(* Logix 5000 project; controller cal1615 1756-L62 rev 20.19; software revision 20.05; part 36 of 82 *)
(* tags used below, declared in another part *)
   AFI : BOOL;   // Always False Bit
   FAULT : BOOL;   // Fault AFI
   p01_recipe_active : recipe;   // Active Recipe
   p01r09_pb_global_reset : BOOL;   // System Modes PB: Global Fault Reset
   p02_dint_from_hmi : hmi_dint;
   p02_real_from_hmi : hmi_real;   // MOP HMI Iface Real from HMI
   p11r31_timer_prs : TIMER;   // Advanced Cooling Pump Pressure On Delay
   p13r30_request_cool : BOOL;   // Zone 3 Temperature Control Request Cooling
   p19_ai_prs : REAL;   // Advanced Cooling Analog Input Pressure [PSI]
   p19_ai_tc01 : REAL;   // Advanced Cooling Analog Input Control Temperature 1
   p19_ao_cv : REAL;   // Advanced Cooling Analog Output Control Valve
   p19_ao_prs_cv : REAL;   // Advanced Cooling Pressure Control AO: Control Value
   p19_di_pump : BOOL;
   p19_di_tc01_bo : BOOL;   // Advanced Cooling Digital Input Control Thermocouple 1 Failure
   p19_do_pump : BOOL;   // Advanced Cooling Digital Output Enable Pump
   p19_param_pid2_ff : REAL;
   p19_param_pid2_kd : REAL;
   p19_param_pid2_ki : REAL;
   p19_param_pid2_kp : REAL;
   p19_param_prs_dev : REAL;
   p19_param_prs_pid_ff : REAL;
   p19_param_prs_pid_kd : REAL;
   p19_param_prs_pid_ki : REAL;
   p19_param_prs_pid_kp : REAL;
   p19_param_tc01_dev : REAL;
   p19_param_zone_pressure : REAL;   // Advanced Cooling Parameter Minimum Pressusre
   p19r01 : routine;   // Advanced Cooling Main
   p19r10 : routine;   // Advanced Cooling Parameters
   p19r10_timer_warning : TIMER[4];   // Advanced Cooling Parameters Warning Delay
   p19r16_pid_temp_cv : DINT;   // Advanced Cooling Temperature Control PID Control Valve
   p19r30 : routine;   // Advanced Cooling Temperature Control
   p19r30_cv_man_sp : REAL;   // Advanced Cooling Manual Control Valve Setpoint
   p19r30_pb_auto : BOOL;   // Advanced Cooling Temmperature Control PB: Zone in Auto
   p19r30_pb_manual : BOOL;   // Advanced Cooling Temmperature Control PB: Zone in Manual
   p19r30_pb_zone_off : BOOL;   // Advanced Cooling Temmperature Control PB: Zone Off
   p19r30_pb_zone_on : BOOL;   // Advanced Cooling Temmperature Control PB: Zone On
   p19r30_permissive_run : BOOL;   // Advanced Cooling Temperature Control Permissive Run
   p19r30_pid_temp : PID;   // Advanced Cooling Temperature Control PID
   p19r30_pid_temp_pv : DINT;   // Advanced Cooling Temperature Control PID Process Variable
   p19r30_pid_temp_sp : DINT;   // Advanced Cooling Temeperature Control PID Setpoint
   p19r30_request_cool : BOOL;   // Advanced Cooling Temperature Control Request Cool
   p19r30_request_manual : BOOL;   // Advanced Cooling Temperature Control Request Manual Control
   p19r30_timer_fault : TIMER[4];   // Advanced Cooling Temperature Control Thermocouple Failure
   p19r30_timer_warning : TIMER[4];   // Advanced Cooling Temperature Control Warning Delay
   p19r31 : routine;   // Advanced Cooling Pump
   p19r31_pb_start : BOOL;   // Advanced Cooling Pump PB: Start pump
   p19r31_pb_stop : BOOL;   // Advanced Cooling Pump PB: Stop Pump
   p19r31_request_a00 : BOOL;   // Advanced Cooling Pump Request Pressure Failure Fault
   p19r31_request_auto_run : BOOL;   // Advanced Cooling Pump Request Auto Run
   p19r31_request_manual_run : BOOL;
   p19r31_run_permissive : BOOL;   // Advanced Cooling Pump Run Permissive
   p19r31_timer_fault : TIMER[4];   // Advanced Cooling Pump Fault Delay
   p19r31_timer_warning : TIMER[4];   // Advanced Cooling Pump Warning Delay
   p19r32 : routine;
   p19r32_cv_man_sp : REAL;
   p19r32_pb_auto : BOOL;   // Advanced Cooling Temmperature Control PB: Zone in Auto
   p19r32_pb_manual : BOOL;   // Advanced Cooling Temmperature Control PB: Zone in Manual
   p19r32_pb_zone_off : BOOL;   // Advanced Cooling Temmperature Control PB: Zone Off
   p19r32_pb_zone_on : BOOL;   // Advanced Cooling Temmperature Control PB: Zone On
   p19r32_permissive_run : BOOL;   // Advanced Cooling Temperature Control Permissive Run
   p19r32_pid_prs : PID;   // Advanced Cooling Temperature Control Pressure Control PID
   p19r32_pid_prs_sp : REAL;   // Advanced Cooling Temmperature Control Pressure Setpoint
   p19r32_pid_temp_cv : REAL;
   p19r32_pid_temp_pv : DINT;   // Advanced Cooling Temperature Control PID Process Variable
   p19r32_request_cool : BOOL;   // Advanced Cooling Temperature Control Request Cool
   p19r32_request_manual : BOOL;   // Advanced Cooling Temperature Control Request Manual Control
   p19r32_timer_fault : TIMER[4];   // Advanced Cooling Pressure Control Fault Dwell Timer
   p19r32_timer_warning : TIMER[4];   // Advanced Cooling Pressure Control Warning Dwell Timer
(* P19_Advanced_Cooling, continued *)

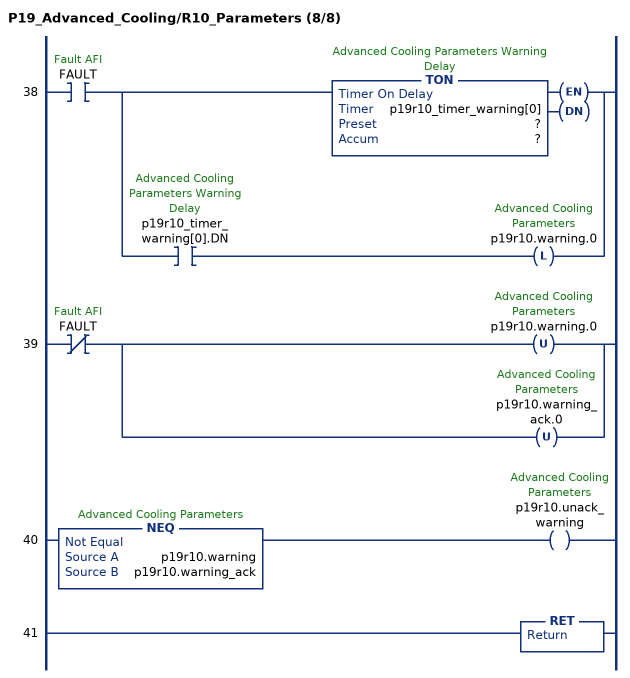
   [picture p656: P19_Advanced_Cooling/R10_Parameters rungs 38-41]
   38: XIC(FAULT)[TON(p19r10_timer_warning[0],?,?) ,XIC(p19r10_timer_warning[0].DN) OTL(p19r10.warning.0) ];
   39: XIO(FAULT)[OTU(p19r10.warning.0) ,OTU(p19r10.warning_ack.0) ];
   40: NEQ(p19r10.warning,p19r10.warning_ack)OTE(p19r10.unack_warning);
   41: RET();
END_ROUTINE

ROUTINE R30_Temperature_Control   (* ladder *)
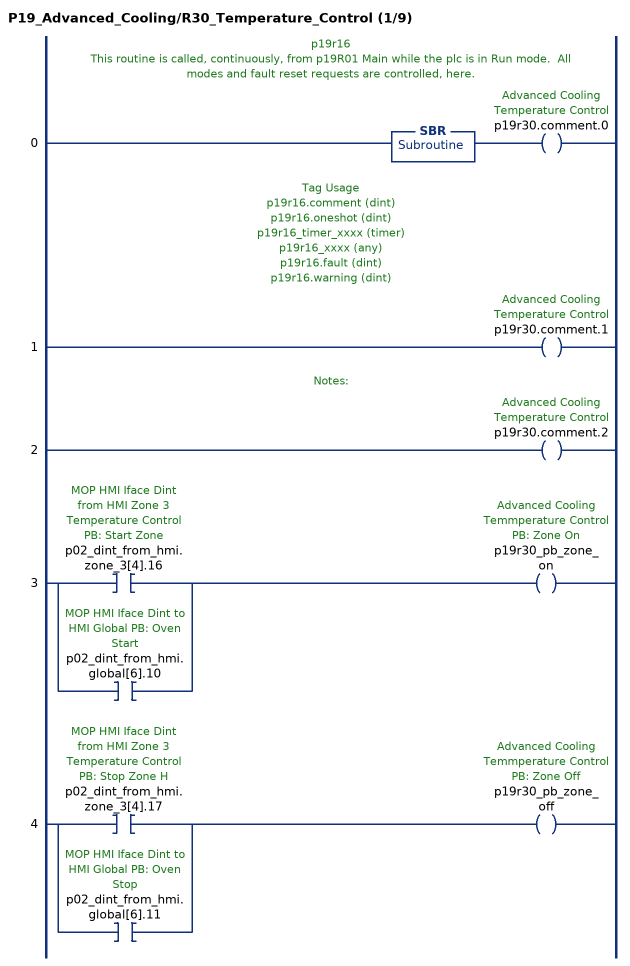
   // p19r16
   // This routine is called, continuously, from p19R01 Main while the plc is in Run mode.  All modes and fault reset requests are controlled, here.
   0: SBR()OTE(p19r30.comment.0);
   // Tag Usage
   // p19r16.comment (dint)
   // p19r16.oneshot (dint)
   // p19r16_timer_xxxx (timer)
   // p19r16_xxxx (any)
   // p19r16.fault (dint)
   // p19r16.warning (dint)
   1: OTE(p19r30.comment.1);
   // Notes:
   2: OTE(p19r30.comment.2);
   3: [XIC(p02_dint_from_hmi.zone_3[4].16) ,XIC(p02_dint_from_hmi.global[6].10) ]OTE(p19r30_pb_zone_on);
   4: [XIC(p02_dint_from_hmi.zone_3[4].17) ,XIC(p02_dint_from_hmi.global[6].11) ]OTE(p19r30_pb_zone_off);
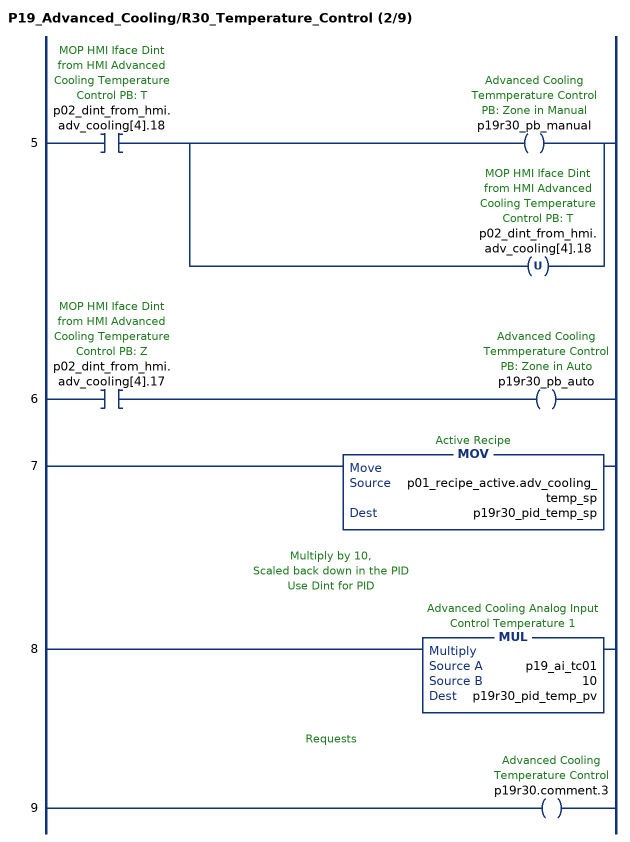
   5: XIC(p02_dint_from_hmi.adv_cooling[4].18)[OTE(p19r30_pb_manual) ,OTU(p02_dint_from_hmi.adv_cooling[4].18) ];
   6: XIC(p02_dint_from_hmi.adv_cooling[4].17)OTE(p19r30_pb_auto);
   7: MOV(p01_recipe_active.adv_cooling_temp_sp,p19r30_pid_temp_sp);
   // Multiply by 10,
   // Scaled back down in the PID
   // Use Dint for PID
   8: MUL(p19_ai_tc01,10,p19r30_pid_temp_pv);
   // Requests
   9: OTE(p19r30.comment.3);
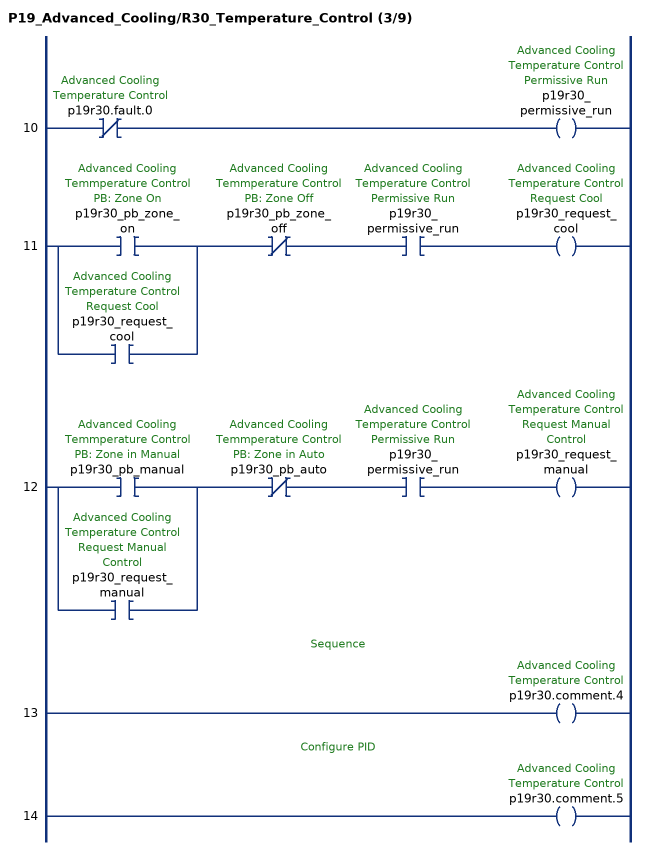
   10: XIO(p19r30.fault.0)OTE(p19r30_permissive_run);
   11: [XIC(p19r30_pb_zone_on) ,XIC(p19r30_request_cool) ]XIO(p19r30_pb_zone_off)XIC(p19r30_permissive_run)OTE(p19r30_request_cool);
   12: [XIC(p19r30_pb_manual) ,XIC(p19r30_request_manual) ]XIO(p19r30_pb_auto)XIC(p19r30_permissive_run)OTE(p19r30_request_manual);
   // Sequence
   13: OTE(p19r30.comment.4);
   // Configure PID
   14: OTE(p19r30.comment.5);
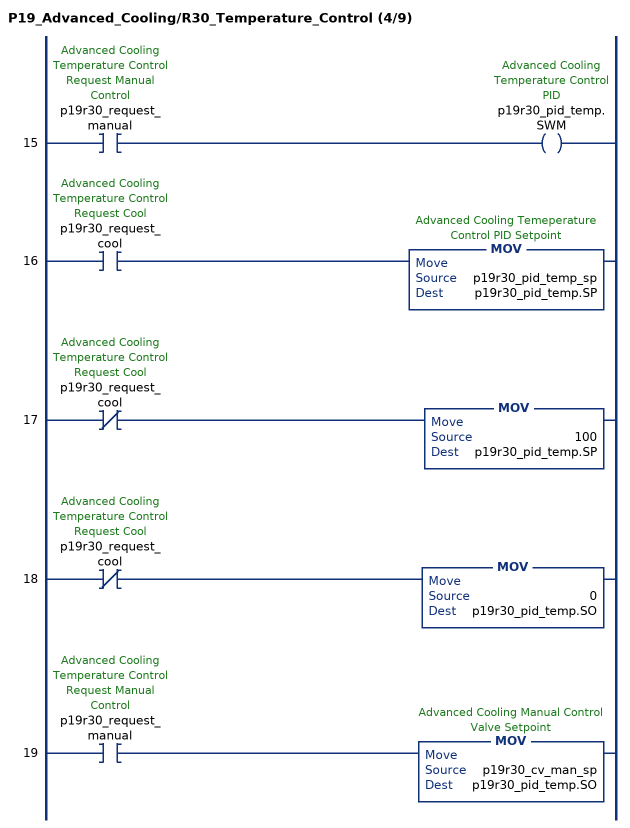
   15: XIC(p19r30_request_manual)OTE(p19r30_pid_temp.SWM);
   16: XIC(p19r30_request_cool)MOV(p19r30_pid_temp_sp,p19r30_pid_temp.SP);
   17: XIO(p19r30_request_cool)MOV(100,p19r30_pid_temp.SP);
   18: XIO(p19r30_request_cool)MOV(0,p19r30_pid_temp.SO);
   19: XIC(p19r30_request_manual)MOV(p19r30_cv_man_sp,p19r30_pid_temp.SO);
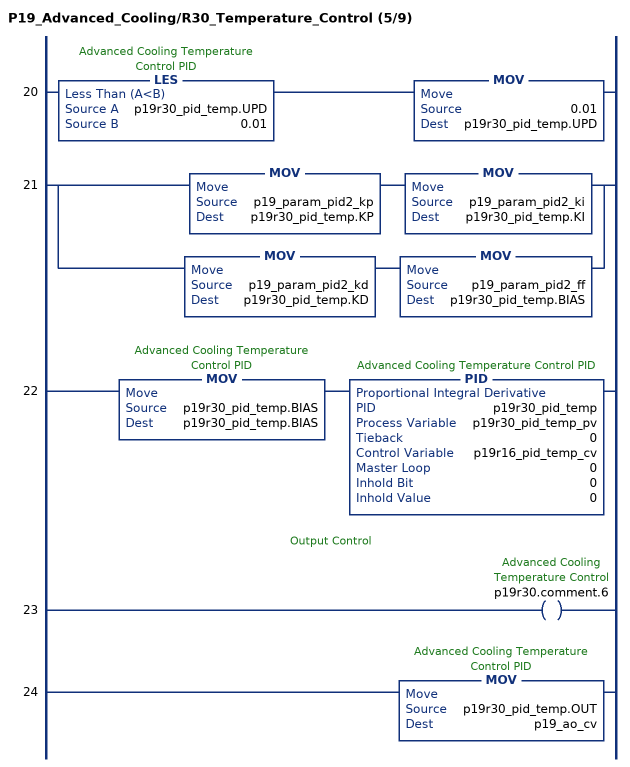
   20: LES(p19r30_pid_temp.UPD,0.01)MOV(0.01,p19r30_pid_temp.UPD);
   21: [MOV(p19_param_pid2_kp,p19r30_pid_temp.KP) MOV(p19_param_pid2_ki,p19r30_pid_temp.KI) ,MOV(p19_param_pid2_kd,p19r30_pid_temp.KD) MOV(p19_param_pid2_ff,p19r30_pid_temp.BIAS) ];
   22: MOV(p19r30_pid_temp.BIAS,p19r30_pid_temp.BIAS)PID(p19r30_pid_temp,p19r30_pid_temp_pv,0,p19r16_pid_temp_cv,0,0,0);
   // Output Control
   23: OTE(p19r30.comment.6);
   24: MOV(p19r30_pid_temp.OUT,p19_ao_cv);
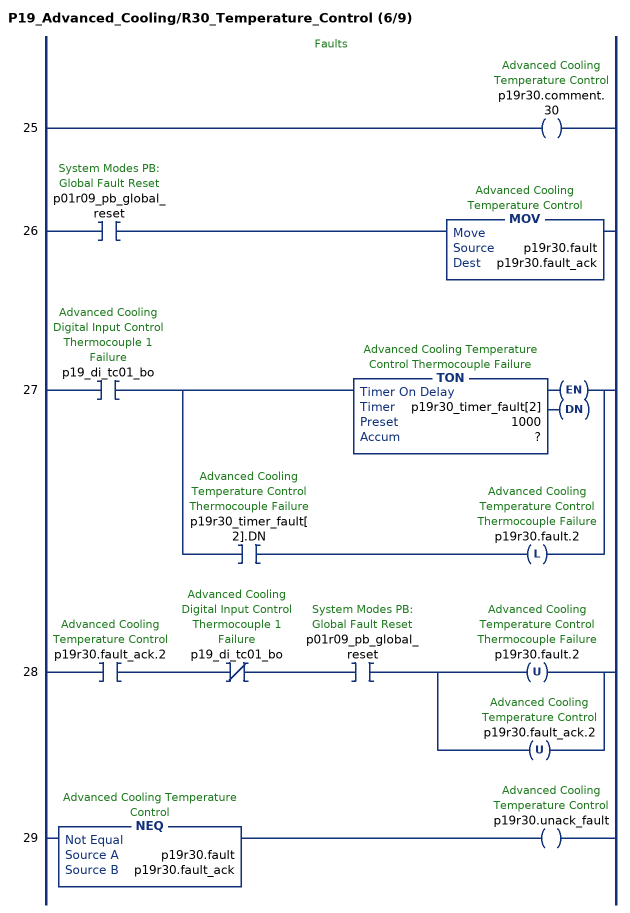
   // Faults
   25: OTE(p19r30.comment.30);
   26: XIC(p01r09_pb_global_reset)MOV(p19r30.fault,p19r30.fault_ack);
   27: XIC(p19_di_tc01_bo)[TON(p19r30_timer_fault[2],?,?) ,XIC(p19r30_timer_fault[2].DN) OTL(p19r30.fault.2) ];
   28: XIC(p19r30.fault_ack.2)XIO(p19_di_tc01_bo)XIC(p01r09_pb_global_reset)[OTU(p19r30.fault.2) ,OTU(p19r30.fault_ack.2) ];
   29: NEQ(p19r30.fault,p19r30.fault_ack)OTE(p19r30.unack_fault);
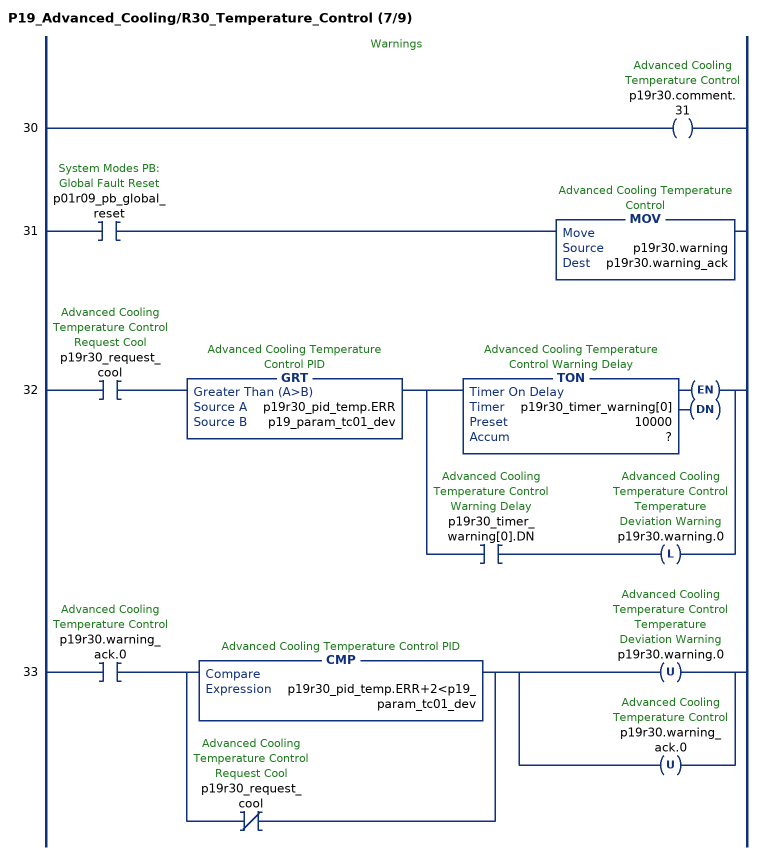
   // Warnings
   30: OTE(p19r30.comment.31);
   31: XIC(p01r09_pb_global_reset)MOV(p19r30.warning,p19r30.warning_ack);
   32: XIC(p19r30_request_cool)GRT(p19r30_pid_temp.ERR,p19_param_tc01_dev)[TON(p19r30_timer_warning[0],?,?) ,XIC(p19r30_timer_warning[0].DN) OTL(p19r30.warning.0) ];
   33: XIC(p19r30.warning_ack.0)[CMP(p19r30_pid_temp.ERR+2<p19_param_tc01_dev) ,XIO(p19r30_request_cool) ][OTU(p19r30.warning.0) ,OTU(p19r30.warning_ack.0) ];
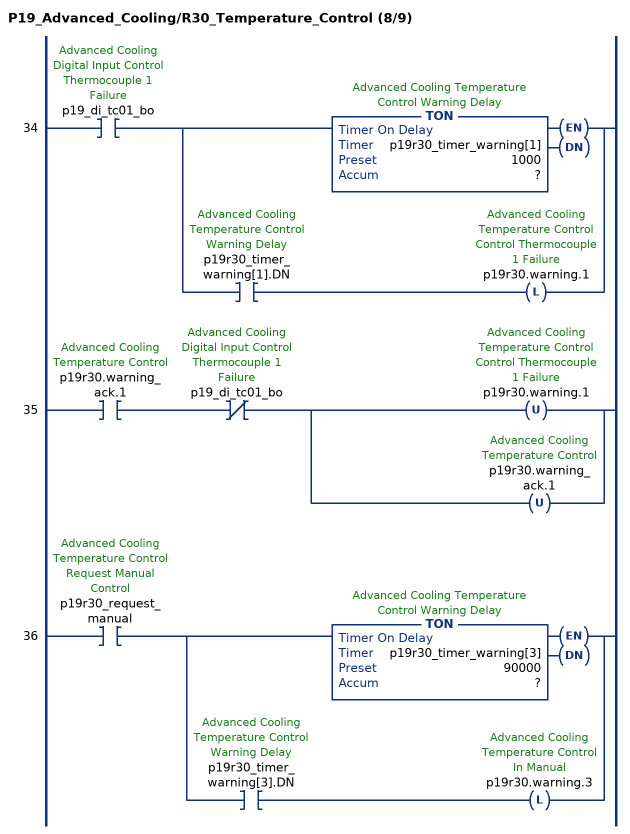
   34: XIC(p19_di_tc01_bo)[TON(p19r30_timer_warning[1],?,?) ,XIC(p19r30_timer_warning[1].DN) OTL(p19r30.warning.1) ];
   35: XIC(p19r30.warning_ack.1)XIO(p19_di_tc01_bo)[OTU(p19r30.warning.1) ,OTU(p19r30.warning_ack.1) ];
   36: XIC(p19r30_request_manual)[TON(p19r30_timer_warning[3],?,?) ,XIC(p19r30_timer_warning[3].DN) OTL(p19r30.warning.3) ];
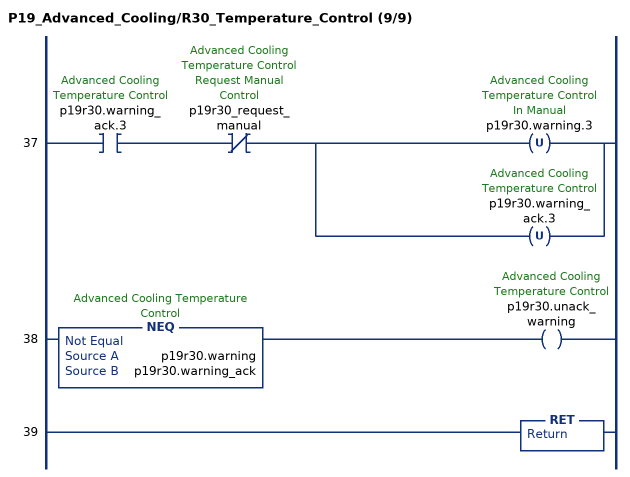
   37: XIC(p19r30.warning_ack.3)XIO(p19r30_request_manual)[OTU(p19r30.warning.3) ,OTU(p19r30.warning_ack.3) ];
   38: NEQ(p19r30.warning,p19r30.warning_ack)OTE(p19r30.unack_warning);
   39: RET();
END_ROUTINE

ROUTINE R31_Pump   (* ladder *)
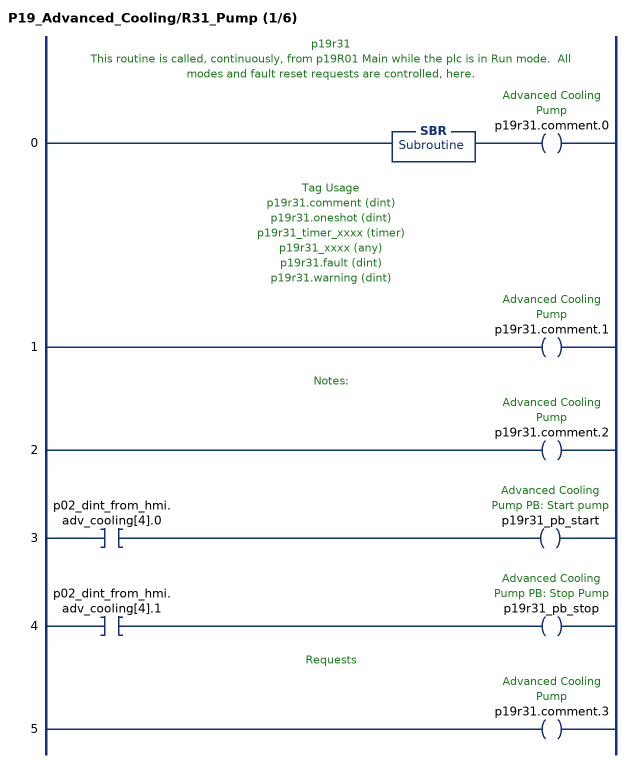
   // p19r31
   // This routine is called, continuously, from p19R01 Main while the plc is in Run mode.  All modes and fault reset requests are controlled, here.
   0: SBR()OTE(p19r31.comment.0);
   // Tag Usage
   // p19r31.comment (dint)
   // p19r31.oneshot (dint)
   // p19r31_timer_xxxx (timer)
   // p19r31_xxxx (any)
   // p19r31.fault (dint)
   // p19r31.warning (dint)
   1: OTE(p19r31.comment.1);
   // Notes:
   2: OTE(p19r31.comment.2);
   3: XIC(p02_dint_from_hmi.adv_cooling[4].0)OTE(p19r31_pb_start);
   4: XIC(p02_dint_from_hmi.adv_cooling[4].1)OTE(p19r31_pb_stop);
   // Requests
   5: OTE(p19r31.comment.3);
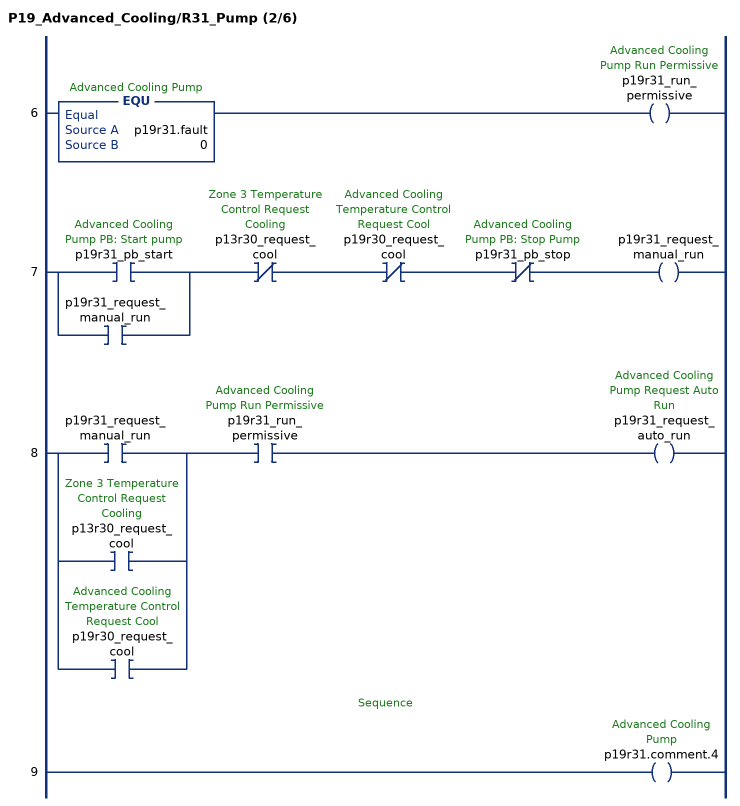
   6: EQU(p19r31.fault,0)OTE(p19r31_run_permissive);
   7: [XIC(p19r31_pb_start) ,XIC(p19r31_request_manual_run) ]XIO(p13r30_request_cool)XIO(p19r30_request_cool)XIO(p19r31_pb_stop)OTE(p19r31_request_manual_run);
   8: [XIC(p19r31_request_manual_run) ,XIC(p13r30_request_cool) ,XIC(p19r30_request_cool) ]XIC(p19r31_run_permissive)OTE(p19r31_request_auto_run);
   // Sequence
   9: OTE(p19r31.comment.4);
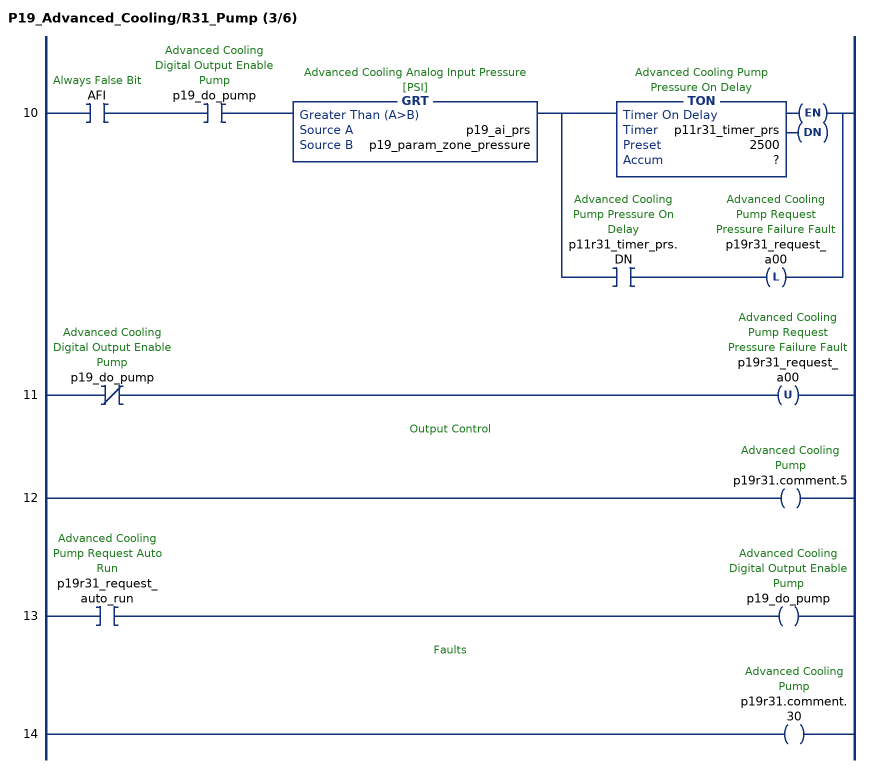
   10: XIC(AFI)XIC(p19_do_pump)GRT(p19_ai_prs,p19_param_zone_pressure)[TON(p11r31_timer_prs,?,?) ,XIC(p11r31_timer_prs.DN) OTL(p19r31_request_a00) ];
   11: XIO(p19_do_pump)OTU(p19r31_request_a00);
   // Output Control
   12: OTE(p19r31.comment.5);
   13: XIC(p19r31_request_auto_run)OTE(p19_do_pump);
   // Faults
   14: OTE(p19r31.comment.30);
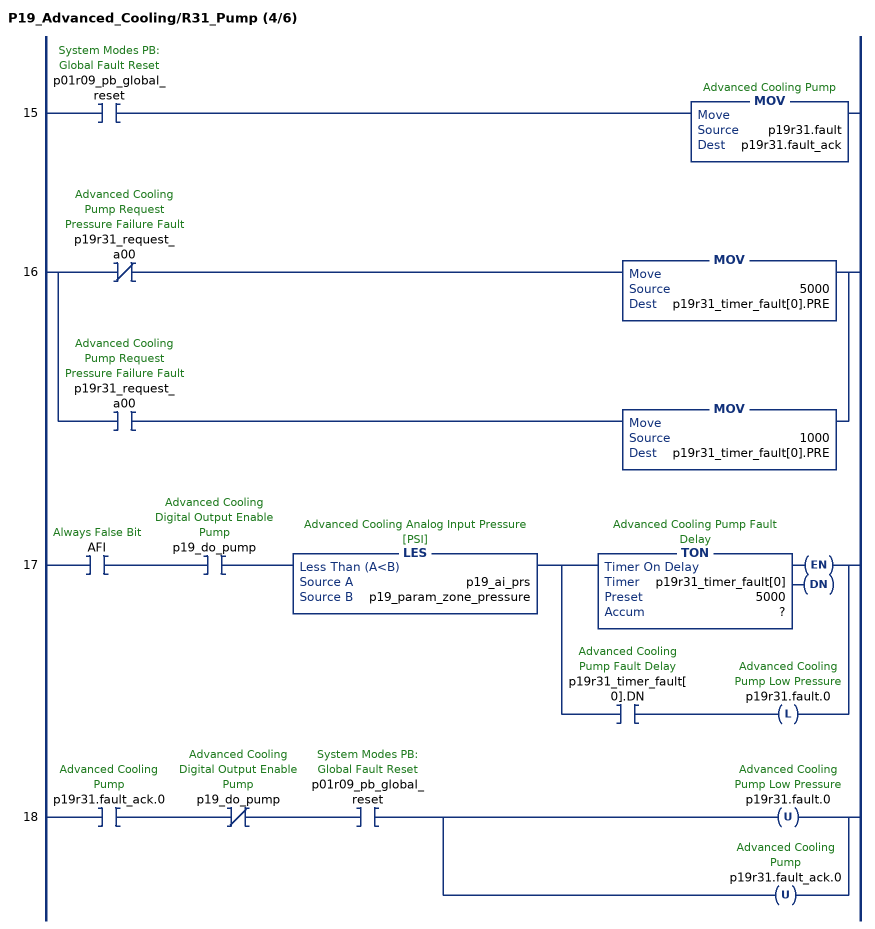
   15: XIC(p01r09_pb_global_reset)MOV(p19r31.fault,p19r31.fault_ack);
   16: [XIO(p19r31_request_a00) MOV(5000,p19r31_timer_fault[0].PRE) ,XIC(p19r31_request_a00) MOV(1000,p19r31_timer_fault[0].PRE) ];
   17: XIC(AFI)XIC(p19_do_pump)LES(p19_ai_prs,p19_param_zone_pressure)[TON(p19r31_timer_fault[0],?,?) ,XIC(p19r31_timer_fault[0].DN) OTL(p19r31.fault.0) ];
   18: XIC(p19r31.fault_ack.0)XIO(p19_do_pump)XIC(p01r09_pb_global_reset)[OTU(p19r31.fault.0) ,OTU(p19r31.fault_ack.0) ];
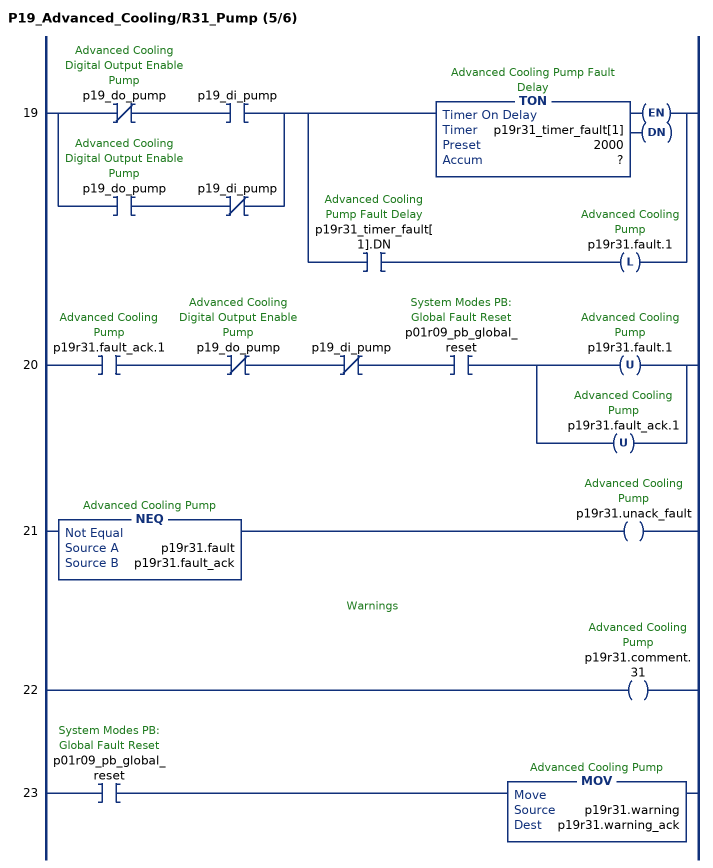
   19: [XIO(p19_do_pump) XIC(p19_di_pump) ,XIC(p19_do_pump) XIO(p19_di_pump) ][TON(p19r31_timer_fault[1],?,?) ,XIC(p19r31_timer_fault[1].DN) OTL(p19r31.fault.1) ];
   20: XIC(p19r31.fault_ack.1)XIO(p19_do_pump)XIO(p19_di_pump)XIC(p01r09_pb_global_reset)[OTU(p19r31.fault.1) ,OTU(p19r31.fault_ack.1) ];
   21: NEQ(p19r31.fault,p19r31.fault_ack)OTE(p19r31.unack_fault);
   // Warnings
   22: OTE(p19r31.comment.31);
   23: XIC(p01r09_pb_global_reset)MOV(p19r31.warning,p19r31.warning_ack);
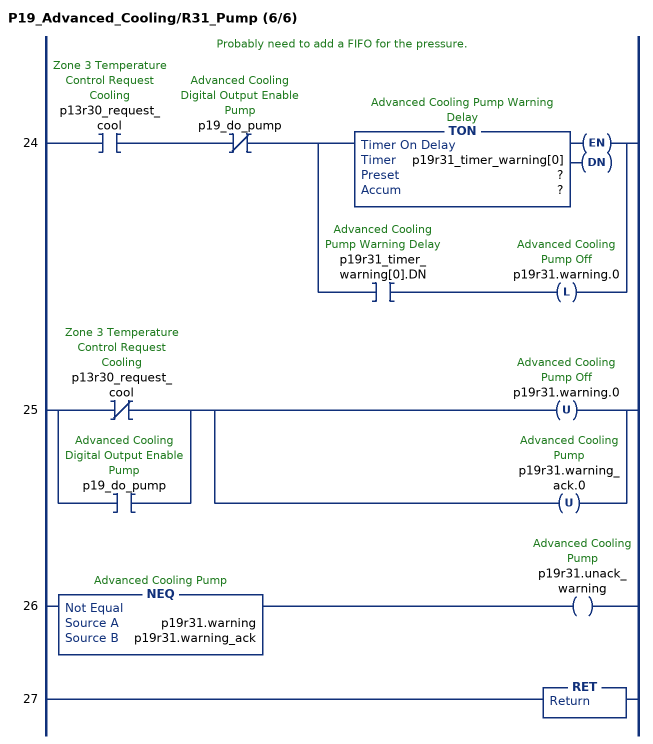
   // Probably need to add a FIFO for the pressure.
   24: XIC(p13r30_request_cool)XIO(p19_do_pump)[TON(p19r31_timer_warning[0],?,?) ,XIC(p19r31_timer_warning[0].DN) OTL(p19r31.warning.0) ];
   25: [XIO(p13r30_request_cool) ,XIC(p19_do_pump) ][OTU(p19r31.warning.0) ,OTU(p19r31.warning_ack.0) ];
   26: NEQ(p19r31.warning,p19r31.warning_ack)OTE(p19r31.unack_warning);
   27: RET();
END_ROUTINE

ROUTINE R32_Pressure_Control   (* ladder *)
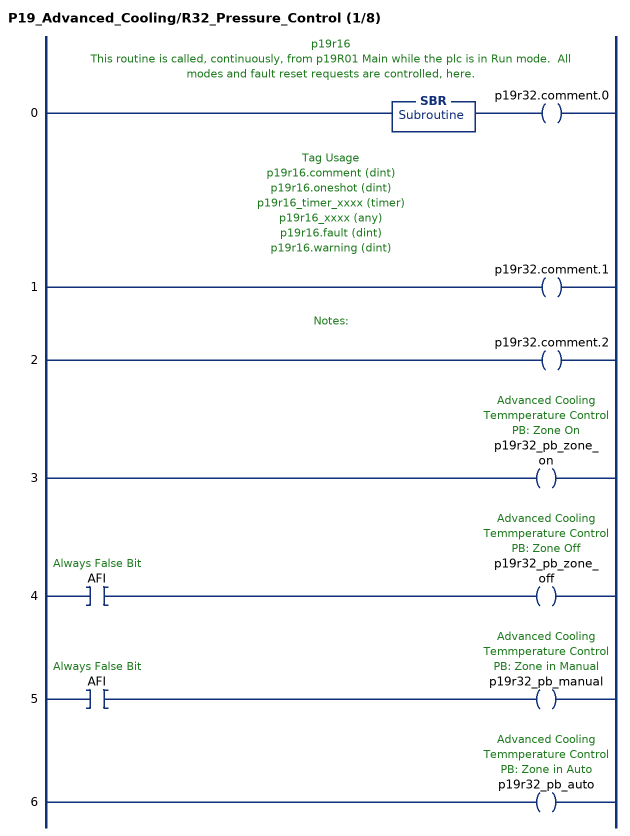
   // p19r16
   // This routine is called, continuously, from p19R01 Main while the plc is in Run mode.  All modes and fault reset requests are controlled, here.
   0: SBR()OTE(p19r32.comment.0);
   // Tag Usage
   // p19r16.comment (dint)
   // p19r16.oneshot (dint)
   // p19r16_timer_xxxx (timer)
   // p19r16_xxxx (any)
   // p19r16.fault (dint)
   // p19r16.warning (dint)
   1: OTE(p19r32.comment.1);
   // Notes:
   2: OTE(p19r32.comment.2);
   3: OTE(p19r32_pb_zone_on);
   4: XIC(AFI)OTE(p19r32_pb_zone_off);
   5: XIC(AFI)OTE(p19r32_pb_manual);
   6: OTE(p19r32_pb_auto);
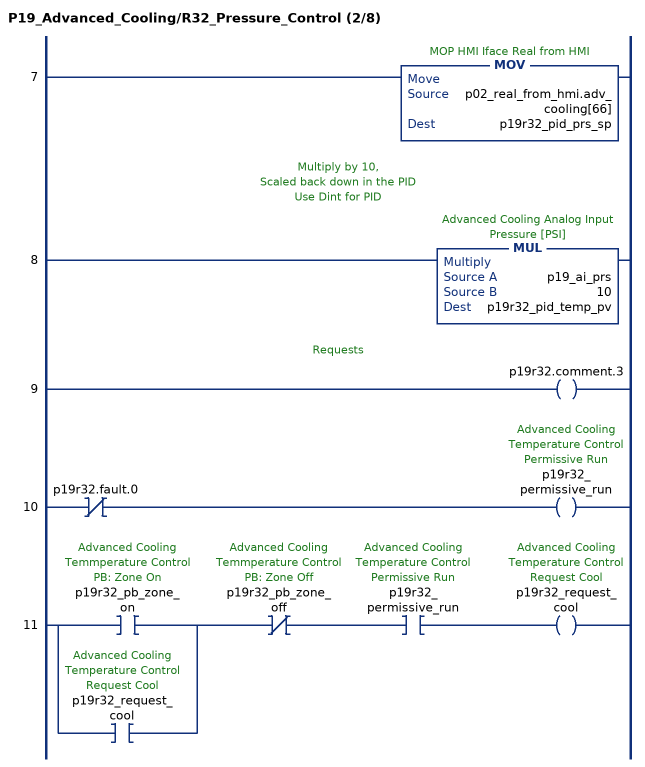
   7: MOV(p02_real_from_hmi.adv_cooling[66],p19r32_pid_prs_sp);
   // Multiply by 10,
   // Scaled back down in the PID
   // Use Dint for PID
   8: MUL(p19_ai_prs,10,p19r32_pid_temp_pv);
   // Requests
   9: OTE(p19r32.comment.3);
   10: XIO(p19r32.fault.0)OTE(p19r32_permissive_run);
   11: [XIC(p19r32_pb_zone_on) ,XIC(p19r32_request_cool) ]XIO(p19r32_pb_zone_off)XIC(p19r32_permissive_run)OTE(p19r32_request_cool);
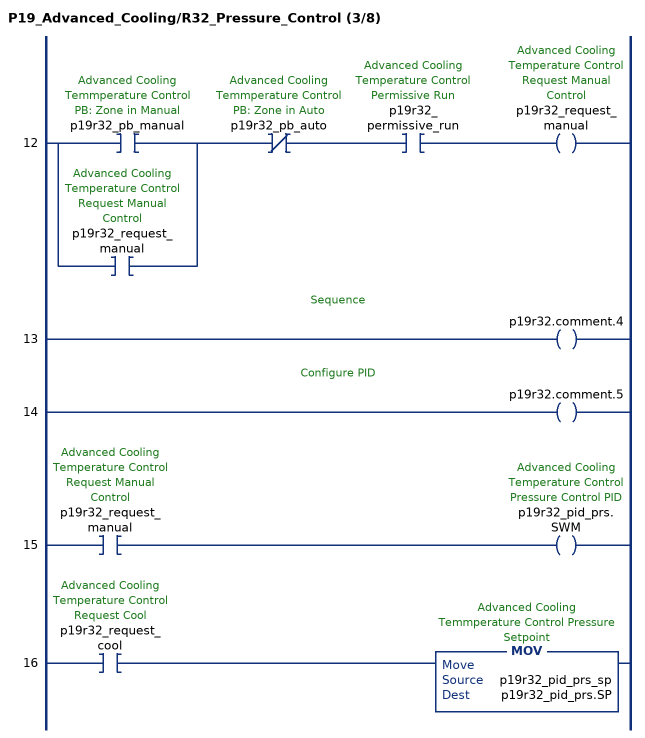
   12: [XIC(p19r32_pb_manual) ,XIC(p19r32_request_manual) ]XIO(p19r32_pb_auto)XIC(p19r32_permissive_run)OTE(p19r32_request_manual);
   // Sequence
   13: OTE(p19r32.comment.4);
   // Configure PID
   14: OTE(p19r32.comment.5);
   15: XIC(p19r32_request_manual)OTE(p19r32_pid_prs.SWM);
   16: XIC(p19r32_request_cool)MOV(p19r32_pid_prs_sp,p19r32_pid_prs.SP);
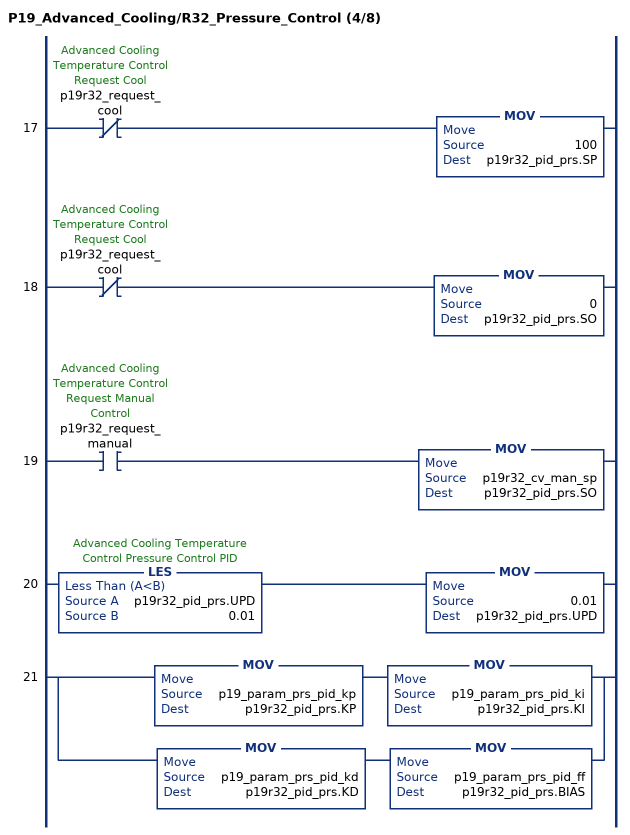
   17: XIO(p19r32_request_cool)MOV(100,p19r32_pid_prs.SP);
   18: XIO(p19r32_request_cool)MOV(0,p19r32_pid_prs.SO);
   19: XIC(p19r32_request_manual)MOV(p19r32_cv_man_sp,p19r32_pid_prs.SO);
   20: LES(p19r32_pid_prs.UPD,0.01)MOV(0.01,p19r32_pid_prs.UPD);
   21: [MOV(p19_param_prs_pid_kp,p19r32_pid_prs.KP) MOV(p19_param_prs_pid_ki,p19r32_pid_prs.KI) ,MOV(p19_param_prs_pid_kd,p19r32_pid_prs.KD) MOV(p19_param_prs_pid_ff,p19r32_pid_prs.BIAS) ];
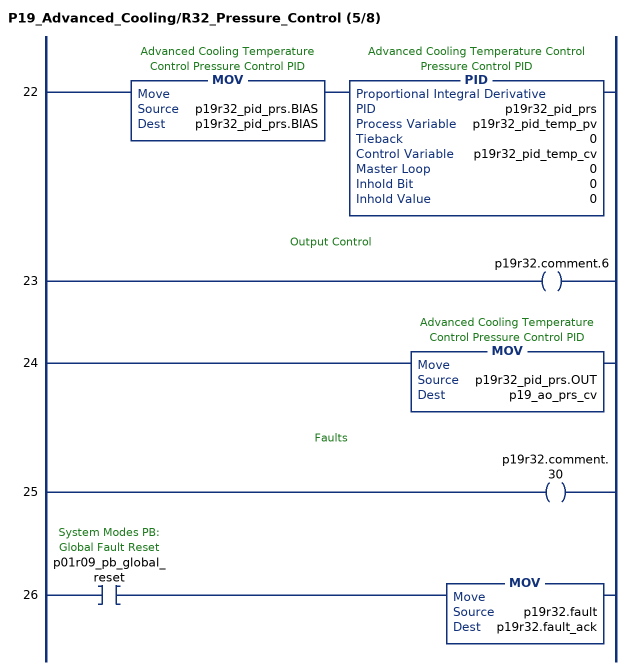
   22: MOV(p19r32_pid_prs.BIAS,p19r32_pid_prs.BIAS)PID(p19r32_pid_prs,p19r32_pid_temp_pv,0,p19r32_pid_temp_cv,0,0,0);
   // Output Control
   23: OTE(p19r32.comment.6);
   24: MOV(p19r32_pid_prs.OUT,p19_ao_prs_cv);
   // Faults
   25: OTE(p19r32.comment.30);
   26: XIC(p01r09_pb_global_reset)MOV(p19r32.fault,p19r32.fault_ack);
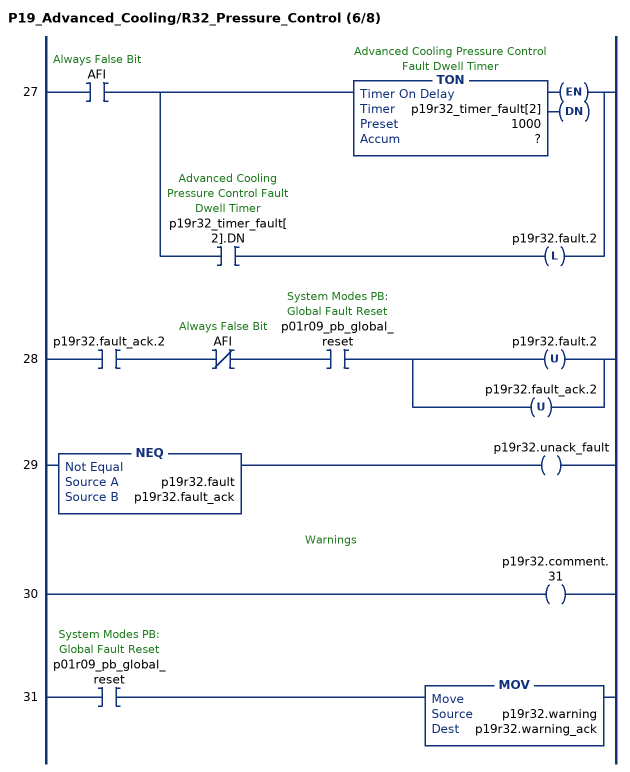
   27: XIC(AFI)[TON(p19r32_timer_fault[2],?,?) ,XIC(p19r32_timer_fault[2].DN) OTL(p19r32.fault.2) ];
   28: XIC(p19r32.fault_ack.2)XIO(AFI)XIC(p01r09_pb_global_reset)[OTU(p19r32.fault.2) ,OTU(p19r32.fault_ack.2) ];
   29: NEQ(p19r32.fault,p19r32.fault_ack)OTE(p19r32.unack_fault);
   // Warnings
   30: OTE(p19r32.comment.31);
   31: XIC(p01r09_pb_global_reset)MOV(p19r32.warning,p19r32.warning_ack);
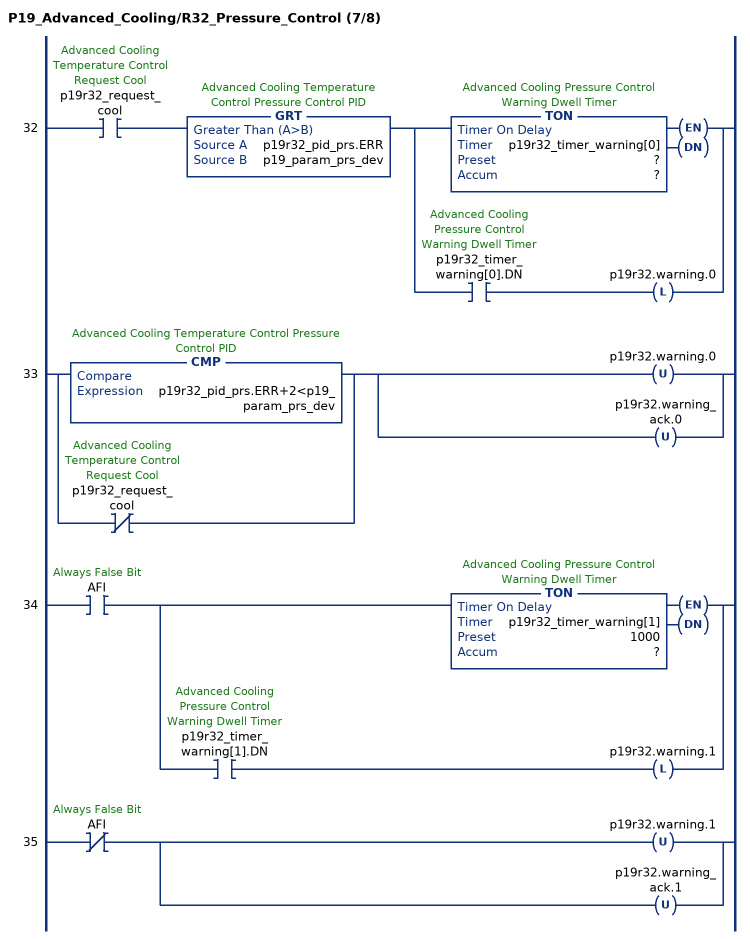
   32: XIC(p19r32_request_cool)GRT(p19r32_pid_prs.ERR,p19_param_prs_dev)[TON(p19r32_timer_warning[0],?,?) ,XIC(p19r32_timer_warning[0].DN) OTL(p19r32.warning.0) ];
   33: [CMP(p19r32_pid_prs.ERR+2<p19_param_prs_dev) ,XIO(p19r32_request_cool) ][OTU(p19r32.warning.0) ,OTU(p19r32.warning_ack.0) ];
   34: XIC(AFI)[TON(p19r32_timer_warning[1],?,?) ,XIC(p19r32_timer_warning[1].DN) OTL(p19r32.warning.1) ];
   35: XIO(AFI)[OTU(p19r32.warning.1) ,OTU(p19r32.warning_ack.1) ];
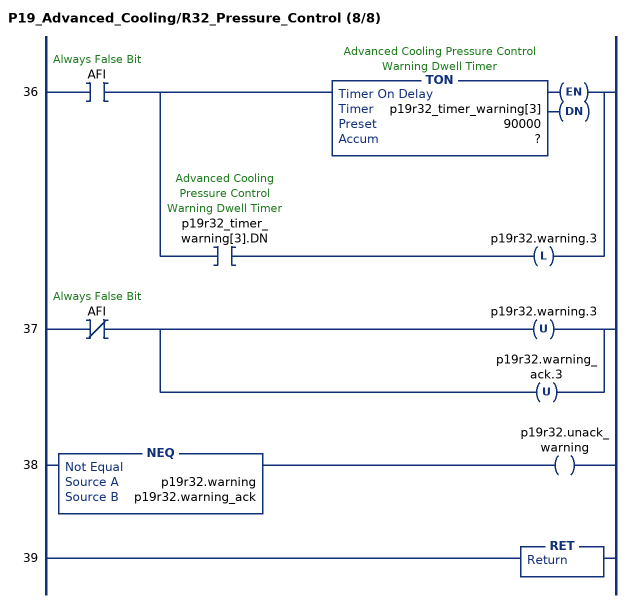
   36: XIC(AFI)[TON(p19r32_timer_warning[3],?,?) ,XIC(p19r32_timer_warning[3].DN) OTL(p19r32.warning.3) ];
   37: XIO(AFI)[OTU(p19r32.warning.3) ,OTU(p19r32.warning_ack.3) ];
   38: NEQ(p19r32.warning,p19r32.warning_ack)OTE(p19r32.unack_warning);
   39: RET();
END_ROUTINE
END_PROGRAM
